Staubli VAL3: trajectory.pjx

--- trajectory.pjx ---
Parameters version=s7.2.1 stackSize=5000 millimeterUnit=true
Program file=computeFrame.pgx
Program file=delete.pgx
Program file=deleteItem.pgx
Program file=duplicate.pgx
Program file=find.pgx
Program file=get.pgx
Program file=getFrame.pgx
Program file=getFrameId.pgx
Program file=getFunctionEdit.pgx
Program file=getFunctionSel.pgx
Program file=getFunctionView.pgx
Program file=getListItem.pgx
Program file=getPoint.pgx
Program file=getSize.pgx
Program file=getSizeItem.pgx
Program file=getTool.pgx
Program file=getTrajItem.pgx
Program file=getTrajType.pgx
Program file=goTo.pgx
Program file=insertItem.pgx
Program file=load.pgx
Program file=loadCycle.pgx
Program file=new.pgx
Program file=onEdit.pgx
Program file=onEditItem.pgx
Program file=onFunctionEdit.pgx
Program file=onFunctionSel.pgx
Program file=onFunctionView.pgx
Program file=onInsert.pgx
Program file=onProgEnd.pgx
Program file=onRun.pgx
Program file=onSave.pgx
Program file=onStart.pgx
Program file=onStop.pgx
Program file=setFrameId.pgx
Program file=setTool.pgx
Program file=setTrajItem.pgx
Data file=trajectory.dtx
Library alias=saveData path=Disk://saveData/saveData.pjx
Library alias=page path=Disk://kernel/template/page/page.pjx
Library alias=use path=Disk://kernel/userPage/userPage.pjx
Type name=TrajectoryItem path=Disk://kernel/template/TrajectoryItem/TrajectoryItem.pjx

--- computeFrame.pgx ---
public program computeFrame(num x_nNewFrame)
begin
end

--- deleteItem.pgx ---
public program deleteItem(num x_nIndex)
begin
end

--- duplicate.pgx ---
public program duplicate(string x_sCopy, string x_sPaste, num& x_nResult[])
  local num i
  local num l_nSize
  local string l_sItem
  local bool l_bFound
  local num l_nResult
begin

end

--- get.pgx ---
public program get(string& x_sItem[], num x_nIndex)
begin

end

--- getFrame.pgx ---
public program getFrame(frame& x_fFrame[], bool x_bCycle)
  local num l_nIndex
begin
end

--- getFunctionSel.pgx ---
public program getFunctionSel(string& x_sName[])
begin
  //
  // define your message for the
  // function KEY
  //
  // NOTE is an ARRAY[0..7]
  //
  // example:
  // x_sName[1]="DEMO"
  // active the F2 button
  //
end

--- getSize.pgx ---
public program getSize(num& x_nSize[])
  local string l_sType
begin
  //
end

--- getSizeItem.pgx ---
public program getSizeItem(bool x_bCycle, num& x_nSize)
  local string l_sType
  local string l_sKey
  local num i
begin
  //
  // get the size of the collection
  //
end

--- getTrajItem.pgx ---
public program getTrajItem(TrajectoryItem& x_tTrajItem[], num x_nIndex)
begin
  //
  // get all the FIELD
  //
  //
  //
end

--- getTrajType.pgx ---
program getTrajType(string& x_sTrajType[])
  local num l_nPos
  local string l_sPath
begin
  // get the trajType
end

--- loadCycle.pgx ---
public program loadCycle(string x_sItem, num& x_nResult[])
begin

end

--- onEdit.pgx ---
public program onEdit(string& x_sItem[])
  local string l_sPath
  local num i
  local string l_sItem
begin
end

--- onEditItem.pgx ---
public program onEditItem(string& x_sEvent[], num x_nIndex, num x_nIndexItem)
begin
  // edit the custom element that was add in the list
end

--- onFunctionSel.pgx ---
public program onFunctionSel(num x_nIndex, string x_sEvent, num x_nFunctionKey)
begin
  //
  // do on Key action
  //
  // x_nIndex = actual index item
  // x_sEvent = actual event item
  //
  switch x_nFunctionKey
    // F1 button
    case 271
    break
    // F2 button
    case 272
    break
    // F3 button
    case 273
    break
    // F4 button
    case 274
    break
    // F5 button
    case 275
    break
    // F6 button
    case 276
    break
    // F7 button
    case 277
    break
    // F8 button
    case 278
    break
  endSwitch
end

--- onInsert.pgx ---
public program onInsert(string& x_sItem[])
  local string l_sEvent
  local num l_nKey
  local num l_nIndex
  local num l_nSize
  local num i
begin
  // get the traj type
end

--- onProgEnd.pgx ---
public program onProgEnd(string& x_sItem[])
begin
end

--- onRun.pgx ---
public program onRun(string& x_sItem[])
begin
end

--- onStop.pgx ---
public program onStop(string& x_sItem[])
begin
end

--- setTool.pgx ---
public program setTool(num x_nIndexGun)
begin
  //
end
